INTERFACE I_Initialisable EXTENDS __SYSTEM.IQueryInterface

METHOD Initialise : HRESULT
VAR_INPUT
END_VAR
END_METHOD

PROPERTY Initialised : BOOL
GET
END_GET
END_PROPERTY

END_INTERFACE

(* stored: Version 1.1.0.1
   Itf I_Initialisable: Id {71ff9433-60c6-4337-b06f-471ab8aac945}
   Method Initialise: Id {5f1fc26c-856c-4028-9354-4db95387c7d5}
   Property Initialised: Id {14e8bd41-19e7-4e4b-8069-6ddf620c91ae}
   Get Get: Id {55314d6c-6e31-4df9-9cee-92d353ca1326} *)
